// TIA Portal V20 export
TYPE "UDT_MTP_BinProcessValueIn"
   STRUCT
      WQC { ExternalWritable := 'False'} : Byte := 16#FF;   // Worst Quality Code CCC
      V : Bool := false;   // External Source Value / Value
      VQC : Byte := 16#FF;   // Quality Code of the current received value
      VState0 { ExternalWritable := 'False'} : String[16] := '';   // Text Replacement Value (False) / text replacement for false
      VState1 { ExternalWritable := 'False'} : String[16] := '';   // Text Replacement Value (True) / text replacement for true
   END_STRUCT;
END_TYPE
